Omron Sysmac Studio project Time_etc (Sysmac Studio 1.65.0.64007, StandardProject)

# Controller new_Controller_0: NX1P2-1040DT1 version 1.69
Task PrimaryTask (priority 4, period or condition 2000): Program0



PROGRAM Program0
VAR
    Start : BOOL;
    Ton : TON;
    Gecen_Sure : LINT;
    Gecen_Sure_INT : ;
    Ton2 : ;
    Ton_ElapsedTime : TIME;
    Ton_2 : TON;
END_VAR

(* Section Section0: ladder, written here as Structured Text *)

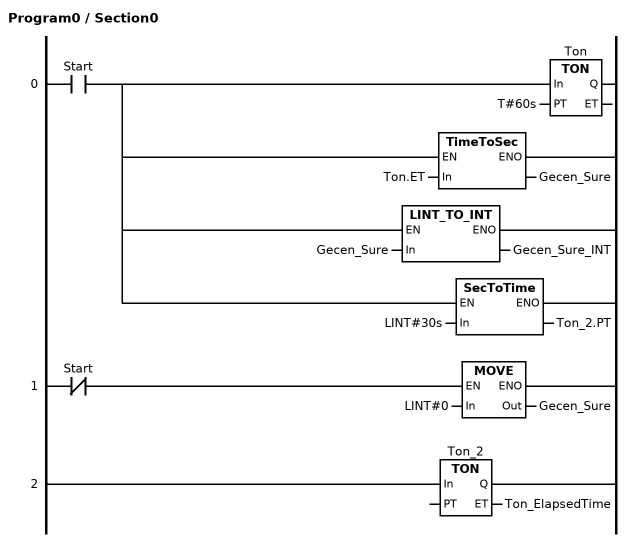
(* Rung 0 *)
Ton(In := Start, PT := T#60s);
IF Start THEN
    Gecen_Sure := TimeToSec(In := Ton.ET);
    Gecen_Sure_INT := LINT_TO_INT(In := Gecen_Sure);
    Ton_2.PT := SecToTime(In := LINT#30s);
END_IF;
(* Rung 1 *)
IF NOT Start THEN Gecen_Sure := LINT#0; END_IF;
(* Rung 2 *)
Ton_2(In := TRUE, ET => Ton_ElapsedTime);
END_PROGRAM